Staubli VAL3: RefreshList.pgx

program RefreshList()
  local num l_ni
begin
  //


end
